PROGRAM MAIN
VAR
END_VAR

MeinProgramm();

END_PROGRAM

(* stored: Version 1.1.0.1, ProductVersion 3.1.4024.5
   POU MAIN: Id {a7fb8e86-b935-41b3-a61d-5c109de02e71}, SpecialFunc None *)
